(* POU RichThreePumpManager, CFC *)
FUNCTION_BLOCK RichThreePumpManager
VAR_INPUT
	start1: BOOL;
	start2: BOOL;
	p1main: BOOL;
	p2main: BOOL;
	p3main: BOOL;
	byCounter: BOOL;
	byWorkTime: BOOL;
	alarm1_in: BOOL;
	alarm2_in: BOOL;
	alarm3_in: BOOL;
	alarmReset: BOOL;
	start1man: BOOL;
	start2man: BOOL;
	start3man: BOOL;
	resetWTone: BOOL;
	resetWTtwo: BOOL;
	resetWTthree: BOOL;
	resetCounterOne: BOOL;
	resetCounterTwo: BOOL;
	resetCounterThree: BOOL;
	delayRepeatedStart: UINT;		(*задержка повторного пуска, сек.*)
	delayStart2: UINT;		(*задержка пуска второго после пуска первого, сек*)
END_VAR
VAR_OUTPUT
	p1mainActive: BOOL;
	p2mainActive: BOOL;
	p3mainActive: BOOL;
	byCounterActive: BOOL;
	byWTactive: BOOL;
	started1: BOOL;
	started2: BOOL;
	started3: BOOL;
	counterOne: UDINT;
	counterTwo: UDINT;
	counterThree: UDINT;
	days1: UINT;
	hours1: UINT;
	minutes1: UINT;
	seconds1: UINT;
	days2: UINT;
	hours2: UINT;
	minutes2: UINT;
	seconds2: UINT;
	days3: UINT;
	hours3: UINT;
	minutes3: UINT;
	seconds3: UINT;
	nextStartP1Timer: UINT;
	nextStartP2Timer: UINT;
	nextStartP3Timer: UINT;
	alarm1active: BOOL;
	alarm2active: BOOL;
	alarm3active: BOOL;
END_VAR
VAR
	ctpr: ChooseThreePumpRegime;
	slft: StartLessFromThree;
	alarmTrig1: RS;
	alarmTrig2: RS;
	alarmTrig3: RS;
	stp: SimpleThreePump;
	frsp1: FastRepeatedStartProtection;
	frsp2: FastRepeatedStartProtection;
	frsp3: FastRepeatedStartProtection;
	pps1: PulsePerSec;
	pps2: PulsePerSec;
	pps3: PulsePerSec;
	icwt1: ImpulsCounter;
	icw2: ImpulsCounter;
	icwt3: ImpulsCounter;
	ts1: TimeSeparator;
	ts2: TimeSeparator;
	ts3: TimeSeparator;
	ic1: ImpulsCounter;
	ic2: ImpulsCounter;
	ic3: ImpulsCounter;
	WorkTimeOne: UDINT;
	WorkTimeTwo: UDINT;
	WorkTimeThree: UDINT;
END_VAR
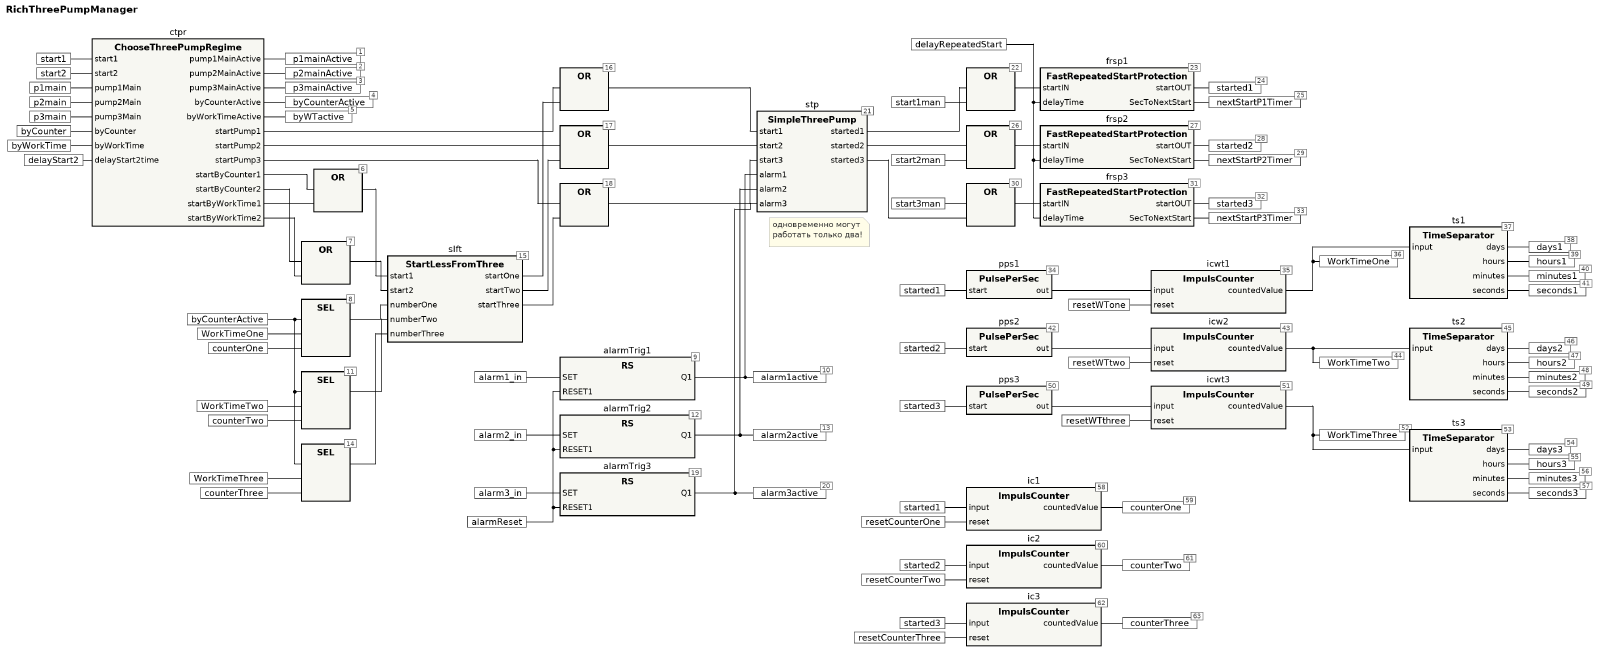
_CFC_ (* Continuous Function Chart, elements in execution order *)
(* одновременно могут / работать только два! *)
#0 ctpr:ChooseThreePumpRegime(start1: start1, start2: start2, pump1Main: p1main, pump2Main: p2main, pump3Main: p3main, byCounter: byCounter, byWorkTime: byWorkTime, delayStart2time: delayStart2)
#1 p1mainActive <= #0.pump1MainActive
#2 p2mainActive <= #0.pump2MainActive
#3 p3mainActive <= #0.pump3MainActive
#4 byCounterActive <= #0.byCounterActive
#5 byWTactive <= #0.byWorkTimeActive
#6 OR(#0.startByCounter1, #0.startByWorkTime1)
#7 OR(#0.startByCounter2, #0.startByWorkTime2)
#8 SEL(byCounterActive, WorkTimeOne, counterOne)
#9 alarmTrig1:RS(SET: alarm1_in, RESET1: alarmReset)
#10 alarm1active <= #9.Q1
#11 SEL(byCounterActive, WorkTimeTwo, counterTwo)
#12 alarmTrig2:RS(SET: alarm2_in, RESET1: alarmReset)
#13 alarm2active <= #12.Q1
#14 SEL(byCounterActive, WorkTimeThree, counterThree)
#15 slft:StartLessFromThree(start1: #6, start2: #7, numberOne: #8, numberTwo: #11, numberThree: #14)
#16 OR(#0.startPump1, #15.startOne)
#17 OR(#0.startPump2, #15.startTwo)
#18 OR(#0.startPump3, #15.startThree)
#19 alarmTrig3:RS(SET: alarm3_in, RESET1: alarmReset)
#20 alarm3active <= #19.Q1
#21 stp:SimpleThreePump(start1: #16, start2: #17, start3: #18, alarm1: #9.Q1, alarm2: #12.Q1, alarm3: #19.Q1)
#22 OR(#21.started1, start1man)
#23 frsp1:FastRepeatedStartProtection(startIN: #22, delayTime: delayRepeatedStart)
#24 started1 <= #23.startOUT
#25 nextStartP1Timer <= #23.SecToNextStart
#26 OR(#21.started2, start2man)
#27 frsp2:FastRepeatedStartProtection(startIN: #26, delayTime: delayRepeatedStart)
#28 started2 <= #27.startOUT
#29 nextStartP2Timer <= #27.SecToNextStart
#30 OR(start3man, #21.started3)
#31 frsp3:FastRepeatedStartProtection(startIN: #30, delayTime: delayRepeatedStart)
#32 started3 <= #31.startOUT
#33 nextStartP3Timer <= #31.SecToNextStart
#34 pps1:PulsePerSec(start: started1)
#35 icwt1:ImpulsCounter(input: #34.out, reset: resetWTone)
#36 WorkTimeOne <= #35.countedValue
#37 ts1:TimeSeparator(input: #35.countedValue)
#38 days1 <= #37.days
#39 hours1 <= #37.hours
#40 minutes1 <= #37.minutes
#41 seconds1 <= #37.seconds
#42 pps2:PulsePerSec(start: started2)
#43 icw2:ImpulsCounter(input: #42.out, reset: resetWTtwo)
#44 WorkTimeTwo <= #43.countedValue
#45 ts2:TimeSeparator(input: #43.countedValue)
#46 days2 <= #45.days
#47 hours2 <= #45.hours
#48 minutes2 <= #45.minutes
#49 seconds2 <= #45.seconds
#50 pps3:PulsePerSec(start: started3)
#51 icwt3:ImpulsCounter(input: #50.out, reset: resetWTthree)
#52 WorkTimeThree <= #51.countedValue
#53 ts3:TimeSeparator(input: #51.countedValue)
#54 days3 <= #53.days
#55 hours3 <= #53.hours
#56 minutes3 <= #53.minutes
#57 seconds3 <= #53.seconds
#58 ic1:ImpulsCounter(input: started1, reset: resetCounterOne)
#59 counterOne <= #58.countedValue
#60 ic2:ImpulsCounter(input: started2, reset: resetCounterTwo)
#61 counterTwo <= #60.countedValue
#62 ic3:ImpulsCounter(input: started3, reset: resetCounterThree)
#63 counterThree <= #62.countedValue
_END_CFC_
(* the same logic as Structured Text *)
(* одновременно могут / работать только два! *)
ctpr(start1 := start1, start2 := start2, pump1Main := p1main, pump2Main := p2main, pump3Main := p3main, byCounter := byCounter, byWorkTime := byWorkTime, delayStart2time := delayStart2);
p1mainActive := ctpr.pump1MainActive;
p2mainActive := ctpr.pump2MainActive;
p3mainActive := ctpr.pump3MainActive;
byCounterActive := ctpr.byCounterActive;
byWTactive := ctpr.byWorkTimeActive;
alarmTrig1(SET := alarm1_in, RESET1 := alarmReset);
alarm1active := alarmTrig1.Q1;
alarmTrig2(SET := alarm2_in, RESET1 := alarmReset);
alarm2active := alarmTrig2.Q1;
slft(start1 := ctpr.startByCounter1 OR ctpr.startByWorkTime1, start2 := ctpr.startByCounter2 OR ctpr.startByWorkTime2, numberOne := SEL(byCounterActive, WorkTimeOne, counterOne), numberTwo := SEL(byCounterActive, WorkTimeTwo, counterTwo), numberThree := SEL(byCounterActive, WorkTimeThree, counterThree));
alarmTrig3(SET := alarm3_in, RESET1 := alarmReset);
alarm3active := alarmTrig3.Q1;
stp(start1 := ctpr.startPump1 OR slft.startOne, start2 := ctpr.startPump2 OR slft.startTwo, start3 := ctpr.startPump3 OR slft.startThree, alarm1 := alarmTrig1.Q1, alarm2 := alarmTrig2.Q1, alarm3 := alarmTrig3.Q1);
frsp1(startIN := stp.started1 OR start1man, delayTime := delayRepeatedStart);
started1 := frsp1.startOUT;
nextStartP1Timer := frsp1.SecToNextStart;
frsp2(startIN := stp.started2 OR start2man, delayTime := delayRepeatedStart);
started2 := frsp2.startOUT;
nextStartP2Timer := frsp2.SecToNextStart;
frsp3(startIN := start3man OR stp.started3, delayTime := delayRepeatedStart);
started3 := frsp3.startOUT;
nextStartP3Timer := frsp3.SecToNextStart;
pps1(start := started1);
icwt1(input := pps1.out, reset := resetWTone);
WorkTimeOne := icwt1.countedValue;
ts1(input := icwt1.countedValue);
days1 := ts1.days;
hours1 := ts1.hours;
minutes1 := ts1.minutes;
seconds1 := ts1.seconds;
pps2(start := started2);
icw2(input := pps2.out, reset := resetWTtwo);
WorkTimeTwo := icw2.countedValue;
ts2(input := icw2.countedValue);
days2 := ts2.days;
hours2 := ts2.hours;
minutes2 := ts2.minutes;
seconds2 := ts2.seconds;
pps3(start := started3);
icwt3(input := pps3.out, reset := resetWTthree);
WorkTimeThree := icwt3.countedValue;
ts3(input := icwt3.countedValue);
days3 := ts3.days;
hours3 := ts3.hours;
minutes3 := ts3.minutes;
seconds3 := ts3.seconds;
ic1(input := started1, reset := resetCounterOne);
counterOne := ic1.countedValue;
ic2(input := started2, reset := resetCounterTwo);
counterTwo := ic2.countedValue;
ic3(input := started3, reset := resetCounterThree);
counterThree := ic3.countedValue;
END_FUNCTION_BLOCK

(* POU StartLessFromThree, ST *)
FUNCTION_BLOCK StartLessFromThree
VAR_INPUT
	start1: BOOL;
	start2: BOOL;
	numberOne: UDINT;
	numberTwo: UDINT;
	numberThree: UDINT;
END_VAR
VAR_OUTPUT
	startOne: BOOL;
	startTwo: BOOL;
	startThree: BOOL;
END_VAR
VAR
	flag1: BOOL := FALSE;
	flag2: BOOL := FALSE;
	starter: UINT;
END_VAR
IF start1 = TRUE THEN

	IF flag1= FALSE THEN

		IF numberOne  <=  numberTwo AND numberOne <= numberThree THEN
			starter := 0;
			flag1 := TRUE;
		END_IF
		
		IF flag1 = FALSE AND  numberTwo  <=  numberOne AND numberTwo <= numberThree THEN
			starter := 1;
			flag1 := TRUE;
		END_IF
		
		IF flag1 = FALSE AND numberThree  <=  numberOne AND numberThree <= numberTwo THEN
			starter := 2;
			flag1 := TRUE;
		END_IF

	END_IF

	CASE starter OF
		0: startOne := TRUE;
		1: startTwo := TRUE;
		2: startThree := TRUE;
	ELSE
		startOne := FALSE;
		startTwo := FALSE;
		startThree := FALSE;
	END_CASE

		IF start2 = TRUE THEN
			IF flag2 = FALSE THEN
				CASE starter OF
					0:   IF numberTwo <= numberThree THEN
							startTwo := TRUE;
							flag2 := TRUE;
						ELSE
							startThree := TRUE;
							flag2 := TRUE;
						END_IF
					1:   IF numberOne <= numberThree THEN
							startOne := TRUE;
							flag2 := TRUE;
						ELSE
							startThree := TRUE;
							flag2 := TRUE;
						END_IF
					2:   IF numberOne <= numberTwo THEN
							startOne := TRUE;
							flag2 := TRUE;
						ELSE
							startTwo := TRUE;
							flag2 := TRUE;
						END_IF
				END_CASE
			END_IF
		ELSE
			CASE starter OF
				0:   startOne := TRUE;
					startTwo := FALSE;
					startThree := FALSE;
					flag2 := FALSE;
				1:   startTwo := TRUE;
					startOne := FALSE;
					startThree := FALSE;
					flag2 := FALSE;
				2:   startThree := TRUE;
					startOne := FALSE;
					startTwo := FALSE;
					flag2 := FALSE;
			ELSE
				startOne := FALSE;
				startTwo := FALSE;
				startThree := FALSE;
	END_CASE
		END_IF

ELSE

		startOne := FALSE;
		startTwo := FALSE;
		startThree := FALSE;
		flag1 := FALSE;

END_IF
END_FUNCTION_BLOCK

(* POU SimpleThreePump, CFC *)
FUNCTION_BLOCK SimpleThreePump
VAR_INPUT
	start1: BOOL; (*сигнал на пуск насоса 1*)
	start2: BOOL; (*сигнал на пуск насоса 2*)
	start3: BOOL; (*сигнал на пуск насоса 3*)
	alarm1: BOOL; (*авария насоса 1*)
	alarm2: BOOL; (*авария насоса 2*)
	alarm3: BOOL; (*авария насоса 3*)
END_VAR
VAR_OUTPUT
	started1: BOOL; (*сигнал на запуск насоса 1*)
	started2: BOOL; (*сигнал на запуск насоса 2*)
	started3: BOOL; (*сигнал на запуск насоса 3*)
END_VAR
VAR
	pump1changer: BOOL;
	pump2changer: BOOL;
	pump3changer: BOOL;
END_VAR
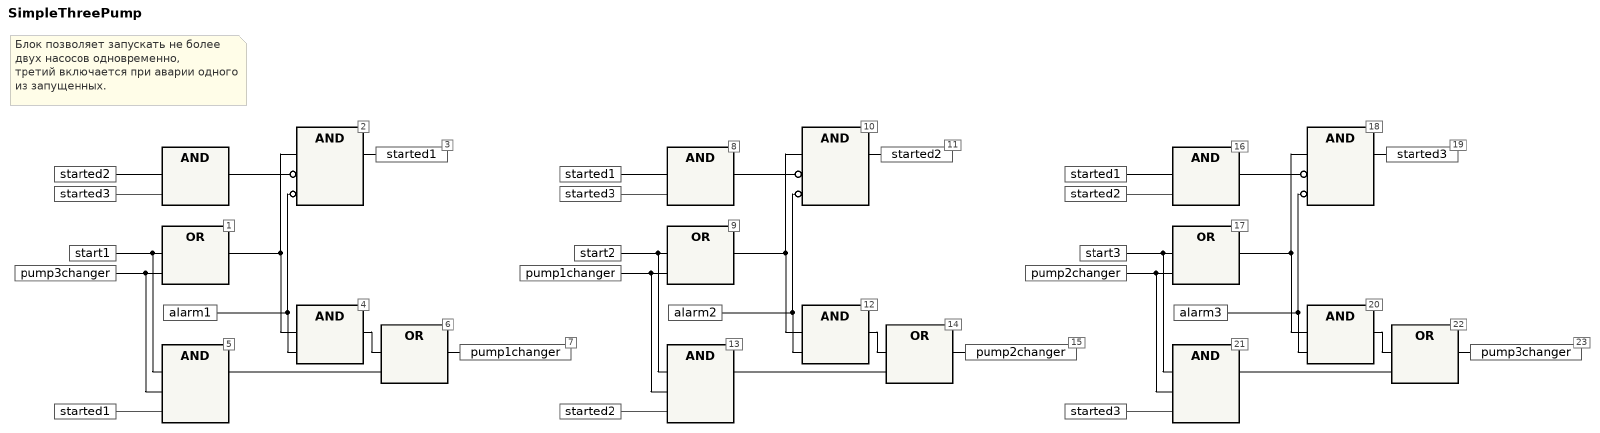
_CFC_ (* Continuous Function Chart, elements in execution order *)
#0 AND(started2, started3)
#1 OR(start1, pump3changer)
(* Блок позволяет запускать не более / двух насосов одновременно, / третий включается при аварии одного / из запущенных. *)
#2 AND(#1, NOT #0, NOT alarm1)
#3 started1 <= #2
#4 AND(#1, alarm1)
#5 AND(start1, pump3changer, started1)
#6 OR(#4, #5)
#7 pump1changer <= #6
#8 AND(started1, started3)
#9 OR(start2, pump1changer)
#10 AND(#9, NOT #8, NOT alarm2)
#11 started2 <= #10
#12 AND(#9, alarm2)
#13 AND(start2, pump1changer, started2)
#14 OR(#12, #13)
#15 pump2changer <= #14
#16 AND(started1, started2)
#17 OR(start3, pump2changer)
#18 AND(#17, NOT #16, NOT alarm3)
#19 started3 <= #18
#20 AND(#17, alarm3)
#21 AND(start3, pump2changer, started3)
#22 OR(#20, #21)
#23 pump3changer <= #22
_END_CFC_
(* the same logic as Structured Text *)
(* Блок позволяет запускать не более / двух насосов одновременно, / третий включается при аварии одного / из запущенных. *)
started1 := (start1 OR pump3changer) AND NOT (started2 AND started3) AND NOT alarm1;
pump1changer := ((start1 OR pump3changer) AND alarm1) OR (start1 AND pump3changer AND started1);
started2 := (start2 OR pump1changer) AND NOT (started1 AND started3) AND NOT alarm2;
pump2changer := ((start2 OR pump1changer) AND alarm2) OR (start2 AND pump1changer AND started2);
started3 := (start3 OR pump2changer) AND NOT (started1 AND started2) AND NOT alarm3;
pump3changer := ((start3 OR pump2changer) AND alarm3) OR (start3 AND pump2changer AND started3);
END_FUNCTION_BLOCK

(* POU TimeSeparator, ST *)
FUNCTION_BLOCK TimeSeparator
VAR_INPUT
	 input: UDINT; (*Вход счетчика  наработки и т.п., сек.*)
END_VAR
VAR_OUTPUT
	days: UINT; (*Выход наработка, дней*)
	hours: UINT; (*Выход наработка, часов*)
	minutes: UINT; (*Выход наработка, минут*)
	seconds: UINT; (*Выход наработка, секунд*)
END_VAR
VAR
	temp: UDINT;
END_VAR
days:= UDINT_TO_INT (input / (60 * 60 * 24));
temp:= input MOD (60 * 60 * 24);
hours:= UDINT_TO_INT (temp / (60 * 60));
temp:= temp MOD (60 * 60);
minutes:= UDINT_TO_INT (temp / 60);
temp:= temp MOD 60;
seconds:= UDINT_TO_INT (temp);
END_FUNCTION_BLOCK

(* POU RichTwoPumpManager, CFC *)
FUNCTION_BLOCK RichTwoPumpManager
VAR_INPUT
	start: BOOL;		(*Сигнал на запуск насоса согласно выбранному режиму.*)
	setPump1main: BOOL;		(*Установить режим - насос 1 = главный.
Включать импульсом.*)
	setPump2main: BOOL;		(*Установить режим - насос 2 = главный.
Включать импульсом.*)
	setByCounter: BOOL;		(*Установить режим - по количеству включений.
Включать импульсом.*)
	setByWorkTime: BOOL;		(*Установить режим - по наработке.
Включать импульсом.*)
	resetPump1counter: BOOL;		(*Сброс счетчика количества включений насоса 1.*)
	resetPump2counter: BOOL;		(*Сброс счетчика количества включений насоса 2.*)
	resetWorkTimePump1: BOOL;		(*Сброс счетчика наработки насоса 1.*)
	resetWorkTimePump2: BOOL;		(*Сброс счетчика наработки насоса 2.*)
	startPump1man: BOOL;		(*Пуск насоса 1 вручную независимо от текущего режима.*)
	startPump2man: BOOL;		(*Пуск насоса 2 вручную независимо от текущего режима.*)
	stop: BOOL;		(*Стоп обоих насосов пока вход активен.
Не стоит применять для штатного останова.*)
	resetAlarms: BOOL;		(*Сброс аварий насоса.*)
	delayRepeatedStartTime: WORD;		(*Количество секунд на задержку повторного пуска насоса.
Защита от частых включений. Если ничего не подключено = 300сек.*)
	alarmPump1input: BOOL;		(*Вход от источника сигнала об аварии насоса 1.*)
	alarmPump2input: BOOL;		(*Вход от источника сигнала об аварии насоса 2.*)
END_VAR
VAR_OUTPUT
	regimePump1Main: BOOL;		(*Текущий режим - насос 1 = главный.*)
	regimePump2Main: BOOL;		(*Текущий режим - насос 2 = главный.*)
	regimeByCounter: BOOL;		(*Текущий режим - по количеству включений.*)
	regimeByWorkTime: BOOL;		(*Текущий режим - по наработке.*)
	counterPump1: DWORD;		(*Количество включений насоса 1.*)
	counterPump2: DWORD;		(*Количество включений насоса 2.*)
	daysPump1: WORD;		(*Количество отработанных дней насоса 1.*)
	hoursPump1: WORD;		(*Количество отработанных часов насоса 1.*)
	minutesPump1: WORD;		(*Количество отработанных минут насоса 1.*)
	secondsPump1: WORD;		(*Количество отработанных секунд насоса 1.*)
	daysPump2: WORD;		(*Количество отработанных дней насоса 2.*)
	hoursPump2: WORD;		(*Количество отработанных часов насоса 2.*)
	minutesPump2: WORD;		(*Количество отработанных минут насоса 2.*)
	secondsPump2: WORD;		(*Количество отработанных секунд насоса 2.*)
	pump1starter: BOOL;		(*Сигнал на запуск насоса 1.*)
	pump2starter: BOOL;		(*Сигнал на запуск насоса 2.*)
	nextStartP1timer: WORD;		(*Обратный отсчет до возможности повторного пуска насоса 1.*)
	nextStartP2timer: WORD;		(*Обратный отсчет до возможности повторного пуска насоса 2.*)
	alarmPump1output: BOOL;		(*Сигнал авария насоса 1.
Триггерится, нужен сброс.*)
	alarmPump2output: BOOL;		(*Сигнал авария насоса 2.
Триггерится, нужен сброс.*)
END_VAR
VAR
	ChoosePumpRegime: ChoosePumpRegime;		(*Блок выбора режима включения.*)
	CounterManager: CounterManager;		(*Блок выбора и запуска насоса по наработке.*)
	WorkTimeManager: WorkTimeManager;		(*Блок выбора и запуска насоса с меньшей наработкой.*)
	simpleTimeManager: SimpleTwoPumpManager;		(*Блок управления двумя насосами, горячий резерв, автоматическое переключение.*)
END_VAR
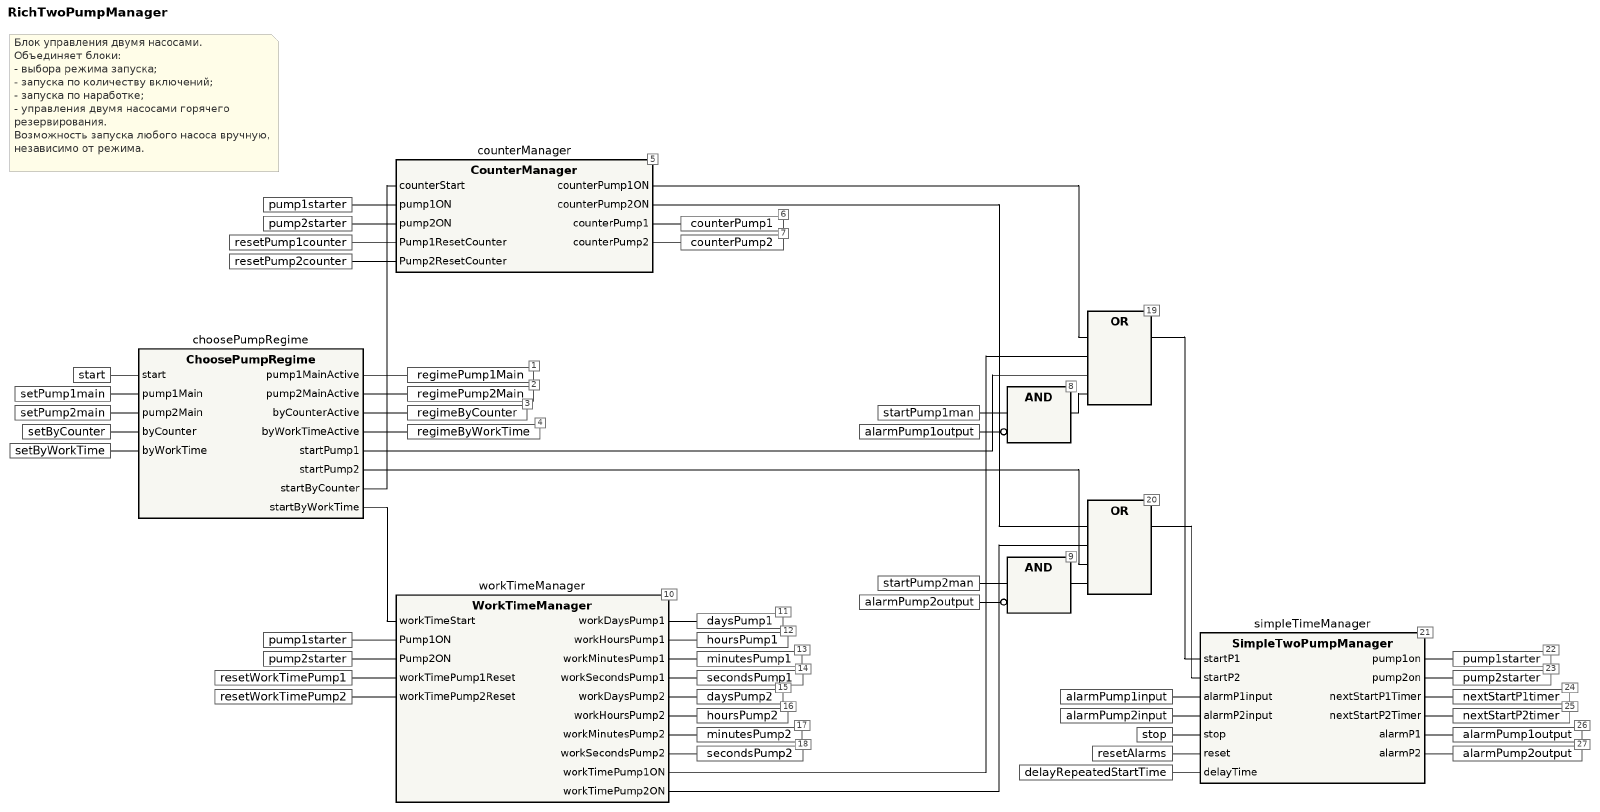
_CFC_ (* Continuous Function Chart, elements in execution order *)
(* Блок управления двумя насосами. / Объединяет блоки: / - выбора режима запуска; / - запуска по количеству включений; / - запуска по наработке; / - управления двумя насосами горячего резервирования. / Возможность запуска любого насоса вручную, / независимо от режима. *)
#0 choosePumpRegime:ChoosePumpRegime(start: start, pump1Main: setPump1main, pump2Main: setPump2main, byCounter: setByCounter, byWorkTime: setByWorkTime)
#1 regimePump1Main <= #0.pump1MainActive
#2 regimePump2Main <= #0.pump2MainActive
#3 regimeByCounter <= #0.byCounterActive
#4 regimeByWorkTime <= #0.byWorkTimeActive
#5 counterManager:CounterManager(counterStart: #0.startByCounter, pump1ON: pump1starter, pump2ON: pump2starter, Pump1ResetCounter: resetPump1counter, Pump2ResetCounter: resetPump2counter)
#6 counterPump1 <= #5.counterPump1
#7 counterPump2 <= #5.counterPump2
#8 AND(startPump1man, NOT alarmPump1output)
#9 AND(startPump2man, NOT alarmPump2output)
#10 workTimeManager:WorkTimeManager(workTimeStart: #0.startByWorkTime, Pump1ON: pump1starter, Pump2ON: pump2starter, workTimePump1Reset: resetWorkTimePump1, workTimePump2Reset: resetWorkTimePump2)
#11 daysPump1 <= #10.workDaysPump1
#12 hoursPump1 <= #10.workHoursPump1
#13 minutesPump1 <= #10.workMinutesPump1
#14 secondsPump1 <= #10.workSecondsPump1
#15 daysPump2 <= #10.workDaysPump2
#16 hoursPump2 <= #10.workHoursPump2
#17 minutesPump2 <= #10.workMinutesPump2
#18 secondsPump2 <= #10.workSecondsPump2
#19 OR(#5.counterPump1ON, #10.workTimePump1ON, #0.startPump1, #8)
#20 OR(#5.counterPump2ON, #10.workTimePump2ON, #0.startPump2, #9)
#21 simpleTimeManager:SimpleTwoPumpManager(startP1: #19, startP2: #20, alarmP1input: alarmPump1input, alarmP2input: alarmPump2input, stop: stop, reset: resetAlarms, delayTime: delayRepeatedStartTime)
#22 pump1starter <= #21.pump1on
#23 pump2starter <= #21.pump2on
#24 nextStartP1timer <= #21.nextStartP1Timer
#25 nextStartP2timer <= #21.nextStartP2Timer
#26 alarmPump1output <= #21.alarmP1
#27 alarmPump2output <= #21.alarmP2
_END_CFC_
(* the same logic as Structured Text *)
(* Блок управления двумя насосами. / Объединяет блоки: / - выбора режима запуска; / - запуска по количеству включений; / - запуска по наработке; / - управления двумя насосами горячего резервирования. / Возможность запуска любого насоса вручную, / независимо от режима. *)
choosePumpRegime(start := start, pump1Main := setPump1main, pump2Main := setPump2main, byCounter := setByCounter, byWorkTime := setByWorkTime);
regimePump1Main := choosePumpRegime.pump1MainActive;
regimePump2Main := choosePumpRegime.pump2MainActive;
regimeByCounter := choosePumpRegime.byCounterActive;
regimeByWorkTime := choosePumpRegime.byWorkTimeActive;
counterManager(counterStart := choosePumpRegime.startByCounter, pump1ON := pump1starter, pump2ON := pump2starter, Pump1ResetCounter := resetPump1counter, Pump2ResetCounter := resetPump2counter);
counterPump1 := counterManager.counterPump1;
counterPump2 := counterManager.counterPump2;
workTimeManager(workTimeStart := choosePumpRegime.startByWorkTime, Pump1ON := pump1starter, Pump2ON := pump2starter, workTimePump1Reset := resetWorkTimePump1, workTimePump2Reset := resetWorkTimePump2);
daysPump1 := workTimeManager.workDaysPump1;
hoursPump1 := workTimeManager.workHoursPump1;
minutesPump1 := workTimeManager.workMinutesPump1;
secondsPump1 := workTimeManager.workSecondsPump1;
daysPump2 := workTimeManager.workDaysPump2;
hoursPump2 := workTimeManager.workHoursPump2;
minutesPump2 := workTimeManager.workMinutesPump2;
secondsPump2 := workTimeManager.workSecondsPump2;
simpleTimeManager(startP1 := counterManager.counterPump1ON OR workTimeManager.workTimePump1ON OR choosePumpRegime.startPump1 OR (startPump1man AND NOT alarmPump1output), startP2 := counterManager.counterPump2ON OR workTimeManager.workTimePump2ON OR choosePumpRegime.startPump2 OR (startPump2man AND NOT alarmPump2output), alarmP1input := alarmPump1input, alarmP2input := alarmPump2input, stop := stop, reset := resetAlarms, delayTime := delayRepeatedStartTime);
pump1starter := simpleTimeManager.pump1on;
pump2starter := simpleTimeManager.pump2on;
nextStartP1timer := simpleTimeManager.nextStartP1Timer;
nextStartP2timer := simpleTimeManager.nextStartP2Timer;
alarmPump1output := simpleTimeManager.alarmP1;
alarmPump2output := simpleTimeManager.alarmP2;
END_FUNCTION_BLOCK

(* POU WorkTimeManager, CFC *)
FUNCTION_BLOCK WorkTimeManager
VAR
	workTimePump1: TimeSeparator;		(*Блок вывода времени наработки  насоса 1.*)
	workTimePump2: TimeSeparator;		(*Блок вывода времени наработки насоса 2.*)
	currentWorkTimePump1: DWORD;		(*Текущая наработка в секундах насоса 1.*)
	currentWorkTimePump2: DWORD;		(*Текущая наработка в секундах насоса 2.*)
	pulsarP1: PulsePerSec;		(*Генератор импульса в секунду для наработки насоса 1.*)
	pulsarP2: PulsePerSec;		(*Генератор импульса в секунду для наработки насоса 2.*)
	timeStartRtrig: R_TRIG;		(*Детектор переднего фронта сигнала на запуск.*)
	timeStartFtrig: F_TRIG;		(*Детектор спада сигнала на запуск.*)
	RStrigTimePump1: RS;		(*RSтриггер сигнала на запуск насоса 1.*)
	RStrigTimePump2: RS;		(*RSтриггер сигнала на запуск насоса 2.*)
END_VAR
VAR_OUTPUT
	workDaysPump1: WORD;		(*Количество отработанных дней для насоса 1.*)
	workHoursPump1: WORD;		(*Количество отработанных часов для насоса 1.*)
	workMinutesPump1: WORD;		(*Количество отработанных минут для насоса 1.*)
	workSecondsPump1: WORD;		(*Количество отработанных секунд для насоса 1.*)
	workDaysPump2: WORD;		(*Количество отработанных дней для насоса 2.*)
	workHoursPump2: WORD;		(*Количество отработанных часов для насоса 2.*)
	workMinutesPump2: WORD;		(*Количество отработанных минут для насоса 2.*)
	workSecondsPump2: WORD;		(*Количество отработанных секунд для насоса 2.*)
	workTimePump1ON: BOOL;		(*Выход на запуск насоса 1.*)
	workTimePump2ON: BOOL;		(*Выход на запуск насоса 2.*)
END_VAR
VAR_INPUT
	workTimeStart: BOOL;		(*Сигнал на запуск насоса с наименьшим временем работы.*)
	Pump1ON: BOOL;		(*Сигнал подтверждение о запуске насоса 1.*)
	Pump2ON: BOOL;		(*Сигнал подтверждение о запуске насоса 2.*)
	workTimePump1Reset: BOOL;		(*Сброс времени наработки насоса 1.*)
	workTimePump2Reset: BOOL;		(*Сброс времени наработки насоса 2.*)
END_VAR
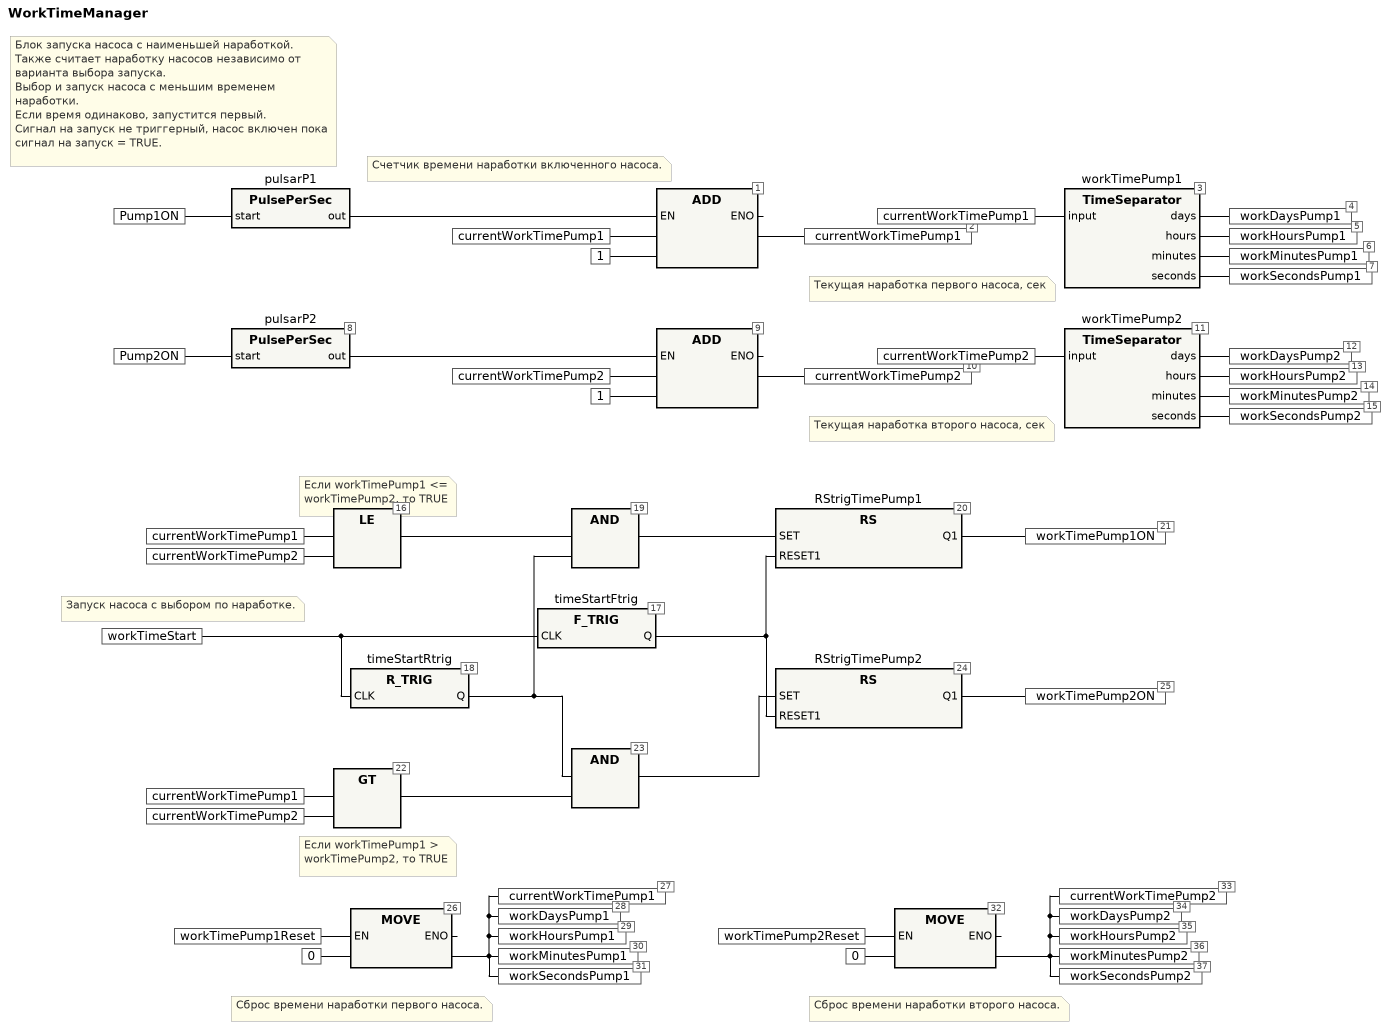
_CFC_ (* Continuous Function Chart, elements in execution order *)
(* Текущая наработка второго насоса, сек *)
(* Сброс времени наработки второго насоса. *)
(* Текущая наработка первого насоса, сек *)
(* Счетчик времени наработки включенного насоса. *)
(* Если workTimePump1 > / workTimePump2, то TRUE *)
(* Если workTimePump1 <= / workTimePump2, то TRUE *)
(* Запуск насоса с выбором по наработке. *)
(* Блок запуска насоса с наименьшей наработкой. / Также считает наработку насосов независимо от варианта выбора запуска. / Выбор и запуск насоса с меньшим временем наработки. / Если время одинаково, запустится первый. / Сигнал на запуск не триггерный, насос включен пока сигнал на запуск = TRUE. *)
(* Сброс времени наработки первого насоса. *)
#0 pulsarP1:PulsePerSec(start: Pump1ON)
#1 ADD(EN: #0.out, currentWorkTimePump1, 1)
#2 currentWorkTimePump1 <= #1
#3 workTimePump1:TimeSeparator(input: currentWorkTimePump1)
#4 workDaysPump1 <= #3.days
#5 workHoursPump1 <= #3.hours
#6 workMinutesPump1 <= #3.minutes
#7 workSecondsPump1 <= #3.seconds
#8 pulsarP2:PulsePerSec(start: Pump2ON)
#9 ADD(EN: #8.out, currentWorkTimePump2, 1)
#10 currentWorkTimePump2 <= #9
#11 workTimePump2:TimeSeparator(input: currentWorkTimePump2)
#12 workDaysPump2 <= #11.days
#13 workHoursPump2 <= #11.hours
#14 workMinutesPump2 <= #11.minutes
#15 workSecondsPump2 <= #11.seconds
#16 LE(currentWorkTimePump1, currentWorkTimePump2)
#17 timeStartFtrig:F_TRIG(CLK: workTimeStart)
#18 timeStartRtrig:R_TRIG(CLK: workTimeStart)
#19 AND(#16, #18.Q)
#20 RStrigTimePump1:RS(SET: #19, RESET1: #17.Q)
#21 workTimePump1ON <= #20.Q1
#22 GT(currentWorkTimePump1, currentWorkTimePump2)
#23 AND(#18.Q, #22)
#24 RStrigTimePump2:RS(SET: #23, RESET1: #17.Q)
#25 workTimePump2ON <= #24.Q1
#26 MOVE(EN: workTimePump1Reset, 0)
#27 currentWorkTimePump1 <= #26
#28 workDaysPump1 <= #26
#29 workHoursPump1 <= #26
#30 workMinutesPump1 <= #26
#31 workSecondsPump1 <= #26
#32 MOVE(EN: workTimePump2Reset, 0)
#33 currentWorkTimePump2 <= #32
#34 workDaysPump2 <= #32
#35 workHoursPump2 <= #32
#36 workMinutesPump2 <= #32
#37 workSecondsPump2 <= #32
_END_CFC_
END_FUNCTION_BLOCK

(* POU SimpleTwoPumpManager, CFC *)
FUNCTION_BLOCK SimpleTwoPumpManager

VAR
	alarmP1trig: RS;		(*Триггер - защелка аварии насоса 1.*)
	alarmP2trig: RS;		(*Триггер - защелка аварии насоса 2.*)
	stopPump1Detector: F_TRIG;		(*Детектор спада сигнала (останов) насоса 1.*)
	stopPump2Detector: F_TRIG;		(*Детектор спада сигнала (останов) насоса 2.*)
	delayAfterStopP2: TOF;		(*Таймер задержки на включение
насоса 1 после останова насоса 2.*)
	delayAfterStopP1: TOF;		(*Таймер задержки на включение
насоса 2 после останова насоса 1.*)
	antiFreqStartPump1: TOF;		(*Таймер - предохранитель от частых пусков насоса 1.*)
	antiFreqStartPump2: TOF;		(*Таймер - предохранитель от частых пусков насоса 2.*)
	startPump1Trig: RS;		(*RS триггер на пуск насоса 1.*)
	startPump2Trig: RS;		(*RS триггер на пуск насоса 2.*)
	stopPump1: F_TRIG;		(*Сигнал на останов насоса 1.*)
	stopPump2: F_TRIG;		(*Сигнал на останов насоса 2.*)
END_VAR
VAR_INPUT
	startP1: BOOL;		(*Сигнал на запуск насоса 1.
Активен - пуск, неактивен - стоп.*)
	startP2: BOOL;		(*Сигнал на запуск насоса 2.
Активен - пуск, неактивен - стоп.*)
	alarmP1input: BOOL;		(*Сигнал авария от насоса 1.*)
	alarmP2input: BOOL;		(*Сигнал авария от насоса 2.*)
	stop: BOOL;		(*Сигнал на останов. Пока активен - пусков нет.
Общий на оба насоса.*)
	reset: BOOL;		(*Сброс аварий.*)
	delayTime: WORD := 300;		(*Задержка на повторный пуск в секундах.
Если ко входу ничего не подключено, то 300сек.*)
END_VAR
VAR_OUTPUT
	pump1on: BOOL;		(*Выход на запуск насоса 1.*)
	pump2on: BOOL;		(*Выход на запуск насоса 2.*)
	nextStartP1Timer: WORD;		(*Счетчик секунд до возможности повторного пуска насоса 1.*)
	nextStartP2Timer: WORD;		(*Счетчик секунд до возможности повторного пуска насоса 2.*)
	alarmP1: BOOL;		(*Статус - авария насоса 1.*)
	alarmP2: BOOL;		(*Статус - авария насоса 2.*)
END_VAR
VAR (* helpers for the ST form of the networks *)
	_t203 : TIME;
END_VAR
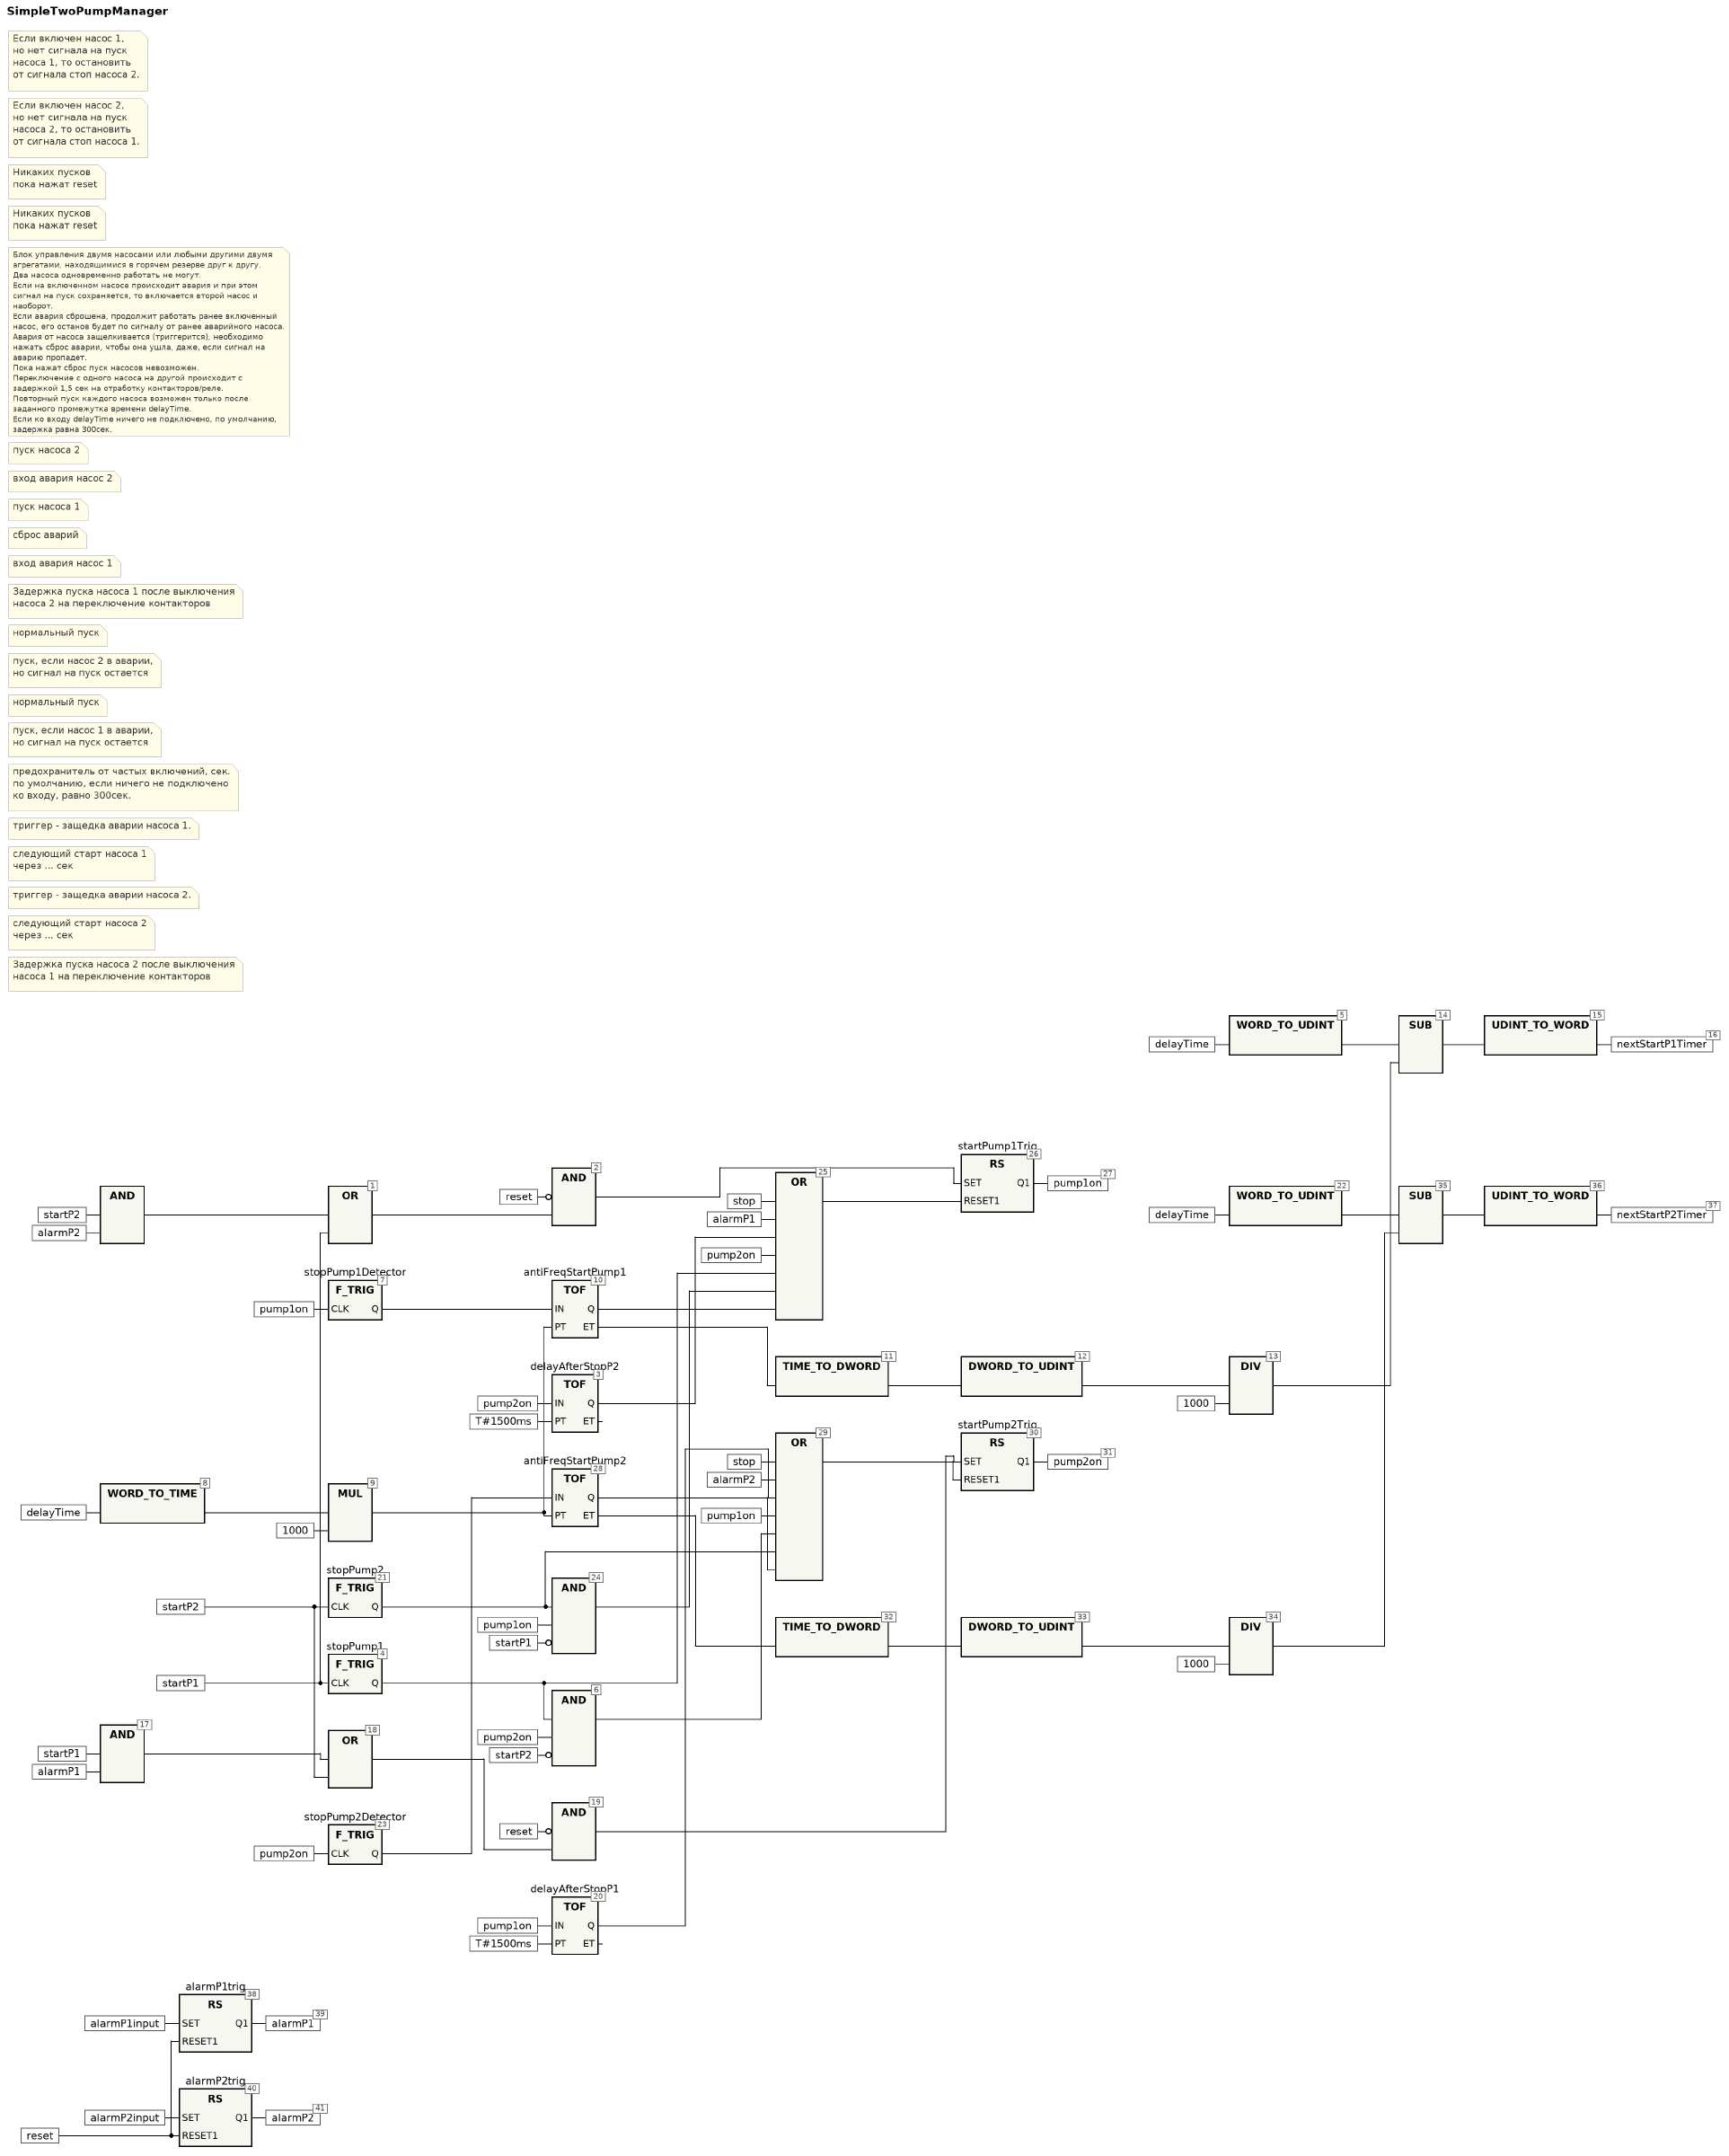
_CFC_ (* Continuous Function Chart, elements in execution order *)
(* Если включен насос 1, / но нет сигнала на пуск / насоса 1, то остановить / от сигнала стоп насоса 2. *)
(* Если включен насос 2, / но нет сигнала на пуск / насоса 2, то остановить / от сигнала стоп насоса 1. *)
(* Никаких пусков / пока нажат reset *)
(* Никаких пусков / пока нажат reset *)
(* Блок управления двумя насосами или любыми другими двумя агрегатами, находящимися в горячем резерве друг к другу. / Два насоса одновременно работать не могут. / Если на включенном насосе происходит авария и при этом сигнал на пуск сохраняется, то включается второй насос и наоборот. / Если авария сброшена, продолжит работать ранее включенный насос, его останов будет по сигналу от ранее аварийного насоса. / Авария от насоса защелкивается (триггерится), необходимо нажать сброс аварии, чтобы она ушла, даже, если сигнал на аварию пропадет. / Пока нажат сброс пуск насосов невозможен. / Переключение с одного насоса на другой происходит с задержкой 1,5 сек на отработку контакторов/реле. / Повторный пуск каждого насоса возможен только после заданного промежутка времени delayTime. / Если ко входу delayTime ничего не подключено, по умолчанию, задержка равна 300сек. *)
(* пуск насоса 2 *)
(* вход авария насос 2 *)
(* пуск насоса 1 *)
(* сброс аварий *)
(* вход авария насос 1 *)
(* Задержка пуска насоса 1 после выключения / насоса 2 на переключение контакторов *)
(* нормальный пуск *)
(* пуск, если насос 2 в аварии, / но сигнал на пуск остается *)
(* нормальный пуск *)
(* пуск, если насос 1 в аварии, / но сигнал на пуск остается *)
(* предохранитель от частых включений, сек. / по умолчанию, если ничего не подключено / ко входу, равно 300сек. *)
(* триггер - защедка аварии насоса 1. *)
(* cледующий старт насоса 1 / через ... сек *)
(* триггер - защедка аварии насоса 2. *)
(* cледующий старт насоса 2 / через ... сек *)
(* Задержка пуска насоса 2 после выключения / насоса 1 на переключение контакторов *)
#0 AND(startP2, alarmP2)
#1 OR(#0, startP1)
#2 AND(NOT reset, #1)
#3 delayAfterStopP2:TOF(IN: pump2on, PT: T#1500ms)
#4 stopPump1:F_TRIG(CLK: startP1)
#5 WORD_TO_UDINT(delayTime)
#6 AND(#4.Q, pump2on, NOT startP2)
#7 stopPump1Detector:F_TRIG(CLK: pump1on)
#8 WORD_TO_TIME(delayTime)
#9 MUL(#8, 1000)
#10 antiFreqStartPump1:TOF(IN: #7.Q, PT: #9)
#11 TIME_TO_DWORD(#10.ET)
#12 DWORD_TO_UDINT(#11)
#13 DIV(#12, 1000)
#14 SUB(#5, #13)
#15 UDINT_TO_WORD(#14)
#16 nextStartP1Timer <= #15
#17 AND(startP1, alarmP1)
#18 OR(#17, startP2)
#19 AND(NOT reset, #18)
#20 delayAfterStopP1:TOF(IN: pump1on, PT: T#1500ms)
#21 stopPump2:F_TRIG(CLK: startP2)
#22 WORD_TO_UDINT(delayTime)
#23 stopPump2Detector:F_TRIG(CLK: pump2on)
#24 AND(#21.Q, pump1on, NOT startP1)
#25 OR(stop, alarmP1, #3.Q, pump2on, #4.Q, #24, #10.Q)
#26 startPump1Trig:RS(SET: #2, RESET1: #25)
#27 pump1on <= #26.Q1
#28 antiFreqStartPump2:TOF(IN: #23.Q, PT: #9)
#29 OR(stop, alarmP2, #20.Q, pump1on, #6, #21.Q, #28.Q)
#30 startPump2Trig:RS(SET: #19, RESET1: #29)
#31 pump2on <= #30.Q1
#32 TIME_TO_DWORD(#28.ET)
#33 DWORD_TO_UDINT(#32)
#34 DIV(#33, 1000)
#35 SUB(#22, #34)
#36 UDINT_TO_WORD(#35)
#37 nextStartP2Timer <= #36
#38 alarmP1trig:RS(SET: alarmP1input, RESET1: reset)
#39 alarmP1 <= #38.Q1
#40 alarmP2trig:RS(SET: alarmP2input, RESET1: reset)
#41 alarmP2 <= #40.Q1
_END_CFC_
(* the same logic as Structured Text *)
(* Если включен насос 1, / но нет сигнала на пуск / насоса 1, то остановить / от сигнала стоп насоса 2. *)
(* Если включен насос 2, / но нет сигнала на пуск / насоса 2, то остановить / от сигнала стоп насоса 1. *)
(* Никаких пусков / пока нажат reset *)
(* Никаких пусков / пока нажат reset *)
(* Блок управления двумя насосами или любыми другими двумя агрегатами, находящимися в горячем резерве друг к другу. / Два насоса одновременно работать не могут. / Если на включенном насосе происходит авария и при этом сигнал на пуск сохраняется, то включается второй насос и наоборот. / Если авария сброшена, продолжит работать ранее включенный насос, его останов будет по сигналу от ранее аварийного насоса. / Авария от насоса защелкивается (триггерится), необходимо нажать сброс аварии, чтобы она ушла, даже, если сигнал на аварию пропадет. / Пока нажат сброс пуск насосов невозможен. / Переключение с одного насоса на другой происходит с задержкой 1,5 сек на отработку контакторов/реле. / Повторный пуск каждого насоса возможен только после заданного промежутка времени delayTime. / Если ко входу delayTime ничего не подключено, по умолчанию, задержка равна 300сек. *)
(* пуск насоса 2 *)
(* вход авария насос 2 *)
(* пуск насоса 1 *)
(* сброс аварий *)
(* вход авария насос 1 *)
(* Задержка пуска насоса 1 после выключения / насоса 2 на переключение контакторов *)
(* нормальный пуск *)
(* пуск, если насос 2 в аварии, / но сигнал на пуск остается *)
(* нормальный пуск *)
(* пуск, если насос 1 в аварии, / но сигнал на пуск остается *)
(* предохранитель от частых включений, сек. / по умолчанию, если ничего не подключено / ко входу, равно 300сек. *)
(* триггер - защедка аварии насоса 1. *)
(* cледующий старт насоса 1 / через ... сек *)
(* триггер - защедка аварии насоса 2. *)
(* cледующий старт насоса 2 / через ... сек *)
(* Задержка пуска насоса 2 после выключения / насоса 1 на переключение контакторов *)
delayAfterStopP2(IN := pump2on, PT := T#1500ms);
stopPump1(CLK := startP1);
stopPump1Detector(CLK := pump1on);
_t203 := WORD_TO_TIME(delayTime) * 1000;
antiFreqStartPump1(IN := stopPump1Detector.Q, PT := _t203);
nextStartP1Timer := UDINT_TO_WORD(WORD_TO_UDINT(delayTime) - (DWORD_TO_UDINT(TIME_TO_DWORD(antiFreqStartPump1.ET)) / 1000));
delayAfterStopP1(IN := pump1on, PT := T#1500ms);
stopPump2(CLK := startP2);
stopPump2Detector(CLK := pump2on);
startPump1Trig(SET := NOT reset AND ((startP2 AND alarmP2) OR startP1), RESET1 := stop OR alarmP1 OR delayAfterStopP2.Q OR pump2on OR stopPump1.Q OR (stopPump2.Q AND pump1on AND NOT startP1) OR antiFreqStartPump1.Q);
pump1on := startPump1Trig.Q1;
antiFreqStartPump2(IN := stopPump2Detector.Q, PT := _t203);
startPump2Trig(SET := NOT reset AND ((startP1 AND alarmP1) OR startP2), RESET1 := stop OR alarmP2 OR delayAfterStopP1.Q OR pump1on OR (stopPump1.Q AND pump2on AND NOT startP2) OR stopPump2.Q OR antiFreqStartPump2.Q);
pump2on := startPump2Trig.Q1;
nextStartP2Timer := UDINT_TO_WORD(WORD_TO_UDINT(delayTime) - (DWORD_TO_UDINT(TIME_TO_DWORD(antiFreqStartPump2.ET)) / 1000));
alarmP1trig(SET := alarmP1input, RESET1 := reset);
alarmP1 := alarmP1trig.Q1;
alarmP2trig(SET := alarmP2input, RESET1 := reset);
alarmP2 := alarmP2trig.Q1;
END_FUNCTION_BLOCK

(* POU TwoPumpOneDriveManager, CFC *)
FUNCTION_BLOCK TwoPumpOneDriveManager
	VAR_INPUT
	start: BOOL;		(*Сигнал на запуск насоса согласно выбранному режиму.*)
	setPump1main: BOOL;		(*Установить режим - насос 1 = главный.
Включать импульсом.*)
	setPump2main: BOOL;		(*Установить режим - насос 2 = главный.
Включать импульсом.*)
	setByCounter: BOOL;		(*Установить режим - по количеству включений.
Включать импульсом.*)
	setByWorkTime: BOOL;		(*Установить режим - по наработке.
Включать импульсом.*)
	resetPump1counter: BOOL;		(*Сброс счетчика количества включений насоса 1.*)
	resetPump2counter: BOOL;		(*Сброс счетчика количества включений насоса 2.*)
	resetWorkTimePump1: BOOL;		(*Сброс счетчика наработки насоса 1.*)
	resetWorkTimePump2: BOOL;		(*Сброс счетчика наработки насоса 2.*)
	startPump1man: BOOL;		(*Пуск насоса 1 вручную независимо от текущего режима.*)
	startPump2man: BOOL;		(*Пуск насоса 2 вручную независимо от текущего режима.*)
	stop: BOOL;		(*Стоп обоих насосов пока вход активен.
Не стоит применять для штатного останова.*)
	resetAlarms: BOOL;		(*Сброс аварий насоса.*)
	delayRepeatedStartTime: WORD;		(*Количество секунд на задержку повторного пуска насоса.
Защита от частых включений. Если ничего не подключено = 300сек.*)
	alarmPump1input: BOOL;		(*Вход от источника сигнала об аварии насоса 1.*)
	alarmPump2input: BOOL;		(*Вход от источника сигнала об аварии насоса 2.*)
	driveAlarm: BOOL;		(*Сигнал авария от ЧРП.*)
END_VAR
VAR_OUTPUT
	regimePump1Main: BOOL;		(*Текущий режим - насос 1 = главный.*)
	regimePump2Main: BOOL;		(*Текущий режим - насос 2 = главный.*)
	regimeByCounter: BOOL;		(*Текущий режим - по количеству включений.*)
	regimeByWorkTime: BOOL;		(*Текущий режим - по наработке.*)
	counterPump1: DWORD;		(*Количество включений насоса 1.*)
	counterPump2: DWORD;		(*Количество включений насоса 2.*)
	daysPump1: WORD;		(*Количество отработанных дней насоса 1.*)
	hoursPump1: WORD;		(*Количество отработанных часов насоса 1.*)
	minutesPump1: WORD;		(*Количество отработанных минут насоса 1.*)
	secondsPump1: WORD;		(*Количество отработанных секунд насоса 1.*)
	daysPump2: WORD;		(*Количество отработанных дней насоса 2.*)
	hoursPump2: WORD;		(*Количество отработанных часов насоса 2.*)
	minutesPump2: WORD;		(*Количество отработанных минут насоса 2.*)
	secondsPump2: WORD;		(*Количество отработанных секунд насоса 2.*)
	drivePower: BOOL;		(*Сигнал на включение контактора частотного преобразователя.*)
	pump1ON: BOOL;		(*Сигнал на включение контактора насоса 1.*)
	pump2ON: BOOL;		(*Сигнал на включение контактора насоса 2.*)
	startDrive: BOOL;		(*Сигнал на запуск в частотный преобразователь.*)
	nextStartP1timer: WORD;		(*Обратный отсчет до возможности повторного пуска насоса 1.*)
	nextStartP2timer: WORD;		(*Обратный отсчет до возможности повторного пуска насоса 2.*)
	alarmPump1output: BOOL;		(*Сигнал авария насоса 1.
Триггерится, нужен сброс.*)
	alarmPump2output: BOOL;		(*Сигнал авария насоса 2.
Триггерится, нужен сброс.*)
END_VAR
VAR

	RichTwoPumpManager: RichTwoPumpManager;		(*Блок управления двумя насосами.*)
	TwoPumpOneDriveModule: TwoPumpOneDriveModule;		(*Модуль управления контакторами двух насосов и питания одного частотного преобразователя.*)
END_VAR
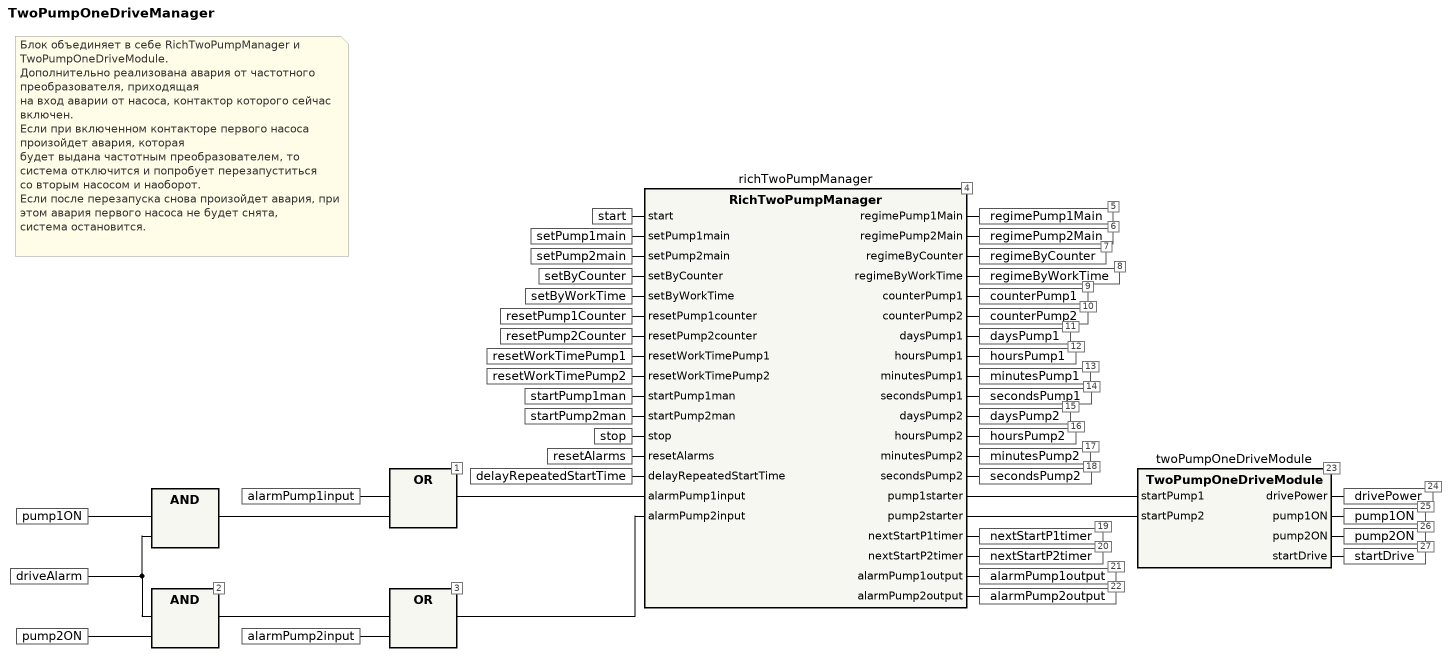
_CFC_ (* Continuous Function Chart, elements in execution order *)
(* Блок объединяет в себе RichTwoPumpManager и TwoPumpOneDriveModule. / Дополнительно реализована авария от частотного преобразователя, приходящая / на вход аварии от насоса, контактор которого сейчас включен. / Если при включенном контакторе первого насоса произойдет авария, которая / будет выдана частотным преобразователем, то система отключится и попробует перезапуститься / со вторым насосом и наоборот. / Если после перезапуска снова произойдет авария, при этом авария первого насоса не будет снята, / система остановится. *)
#0 AND(pump1ON, driveAlarm)
#1 OR(alarmPump1input, #0)
#2 AND(driveAlarm, pump2ON)
#3 OR(#2, alarmPump2input)
#4 richTwoPumpManager:RichTwoPumpManager(start: start, setPump1main: setPump1main, setPump2main: setPump2main, setByCounter: setByCounter, setByWorkTime: setByWorkTime, resetPump1counter: resetPump1Counter, resetPump2counter: resetPump2Counter, resetWorkTimePump1: resetWorkTimePump1, resetWorkTimePump2: resetWorkTimePump2, startPump1man: startPump1man, startPump2man: startPump2man, stop: stop, resetAlarms: resetAlarms, delayRepeatedStartTime: delayRepeatedStartTime, alarmPump1input: #1, alarmPump2input: #3)
#5 regimePump1Main <= #4.regimePump1Main
#6 regimePump2Main <= #4.regimePump2Main
#7 regimeByCounter <= #4.regimeByCounter
#8 regimeByWorkTime <= #4.regimeByWorkTime
#9 counterPump1 <= #4.counterPump1
#10 counterPump2 <= #4.counterPump2
#11 daysPump1 <= #4.daysPump1
#12 hoursPump1 <= #4.hoursPump1
#13 minutesPump1 <= #4.minutesPump1
#14 secondsPump1 <= #4.secondsPump1
#15 daysPump2 <= #4.daysPump2
#16 hoursPump2 <= #4.hoursPump2
#17 minutesPump2 <= #4.minutesPump2
#18 secondsPump2 <= #4.secondsPump2
#19 nextStartP1timer <= #4.nextStartP1timer
#20 nextStartP2timer <= #4.nextStartP2timer
#21 alarmPump1output <= #4.alarmPump1output
#22 alarmPump2output <= #4.alarmPump2output
#23 twoPumpOneDriveModule:TwoPumpOneDriveModule(startPump1: #4.pump1starter, startPump2: #4.pump2starter)
#24 drivePower <= #23.drivePower
#25 pump1ON <= #23.pump1ON
#26 pump2ON <= #23.pump2ON
#27 startDrive <= #23.startDrive
_END_CFC_
(* the same logic as Structured Text *)
(* Блок объединяет в себе RichTwoPumpManager и TwoPumpOneDriveModule. / Дополнительно реализована авария от частотного преобразователя, приходящая / на вход аварии от насоса, контактор которого сейчас включен. / Если при включенном контакторе первого насоса произойдет авария, которая / будет выдана частотным преобразователем, то система отключится и попробует перезапуститься / со вторым насосом и наоборот. / Если после перезапуска снова произойдет авария, при этом авария первого насоса не будет снята, / система остановится. *)
richTwoPumpManager(start := start, setPump1main := setPump1main, setPump2main := setPump2main, setByCounter := setByCounter, setByWorkTime := setByWorkTime, resetPump1counter := resetPump1Counter, resetPump2counter := resetPump2Counter, resetWorkTimePump1 := resetWorkTimePump1, resetWorkTimePump2 := resetWorkTimePump2, startPump1man := startPump1man, startPump2man := startPump2man, stop := stop, resetAlarms := resetAlarms, delayRepeatedStartTime := delayRepeatedStartTime, alarmPump1input := alarmPump1input OR (pump1ON AND driveAlarm), alarmPump2input := (driveAlarm AND pump2ON) OR alarmPump2input);
regimePump1Main := richTwoPumpManager.regimePump1Main;
regimePump2Main := richTwoPumpManager.regimePump2Main;
regimeByCounter := richTwoPumpManager.regimeByCounter;
regimeByWorkTime := richTwoPumpManager.regimeByWorkTime;
counterPump1 := richTwoPumpManager.counterPump1;
counterPump2 := richTwoPumpManager.counterPump2;
daysPump1 := richTwoPumpManager.daysPump1;
hoursPump1 := richTwoPumpManager.hoursPump1;
minutesPump1 := richTwoPumpManager.minutesPump1;
secondsPump1 := richTwoPumpManager.secondsPump1;
daysPump2 := richTwoPumpManager.daysPump2;
hoursPump2 := richTwoPumpManager.hoursPump2;
minutesPump2 := richTwoPumpManager.minutesPump2;
secondsPump2 := richTwoPumpManager.secondsPump2;
nextStartP1timer := richTwoPumpManager.nextStartP1timer;
nextStartP2timer := richTwoPumpManager.nextStartP2timer;
alarmPump1output := richTwoPumpManager.alarmPump1output;
alarmPump2output := richTwoPumpManager.alarmPump2output;
twoPumpOneDriveModule(startPump1 := richTwoPumpManager.pump1starter, startPump2 := richTwoPumpManager.pump2starter);
drivePower := twoPumpOneDriveModule.drivePower;
pump1ON := twoPumpOneDriveModule.pump1ON;
pump2ON := twoPumpOneDriveModule.pump2ON;
startDrive := twoPumpOneDriveModule.startDrive;
END_FUNCTION_BLOCK

(* POU TwoPumpOneDriveModule, CFC *)
FUNCTION_BLOCK TwoPumpOneDriveModule
VAR_INPUT
	startPump1: BOOL;		(*Входящий сигнал на запуск первого насоса.*)
	startPump2: BOOL;		(*Входящий сигнал на запуск второго насоса.*)
END_VAR
VAR_OUTPUT
	drivePower: BOOL;		(*Выход управления контактором питания ЧРП.*)
	pump1ON: BOOL;		(*Выход управления контактором питания насоса 1.*)
	pump2ON: BOOL;		(*Выход управления контактором питания насоса 2.*)
	startDrive: BOOL;		(*Сигнал пуск в ЧРП.*)
END_VAR
VAR
	pump1Off: BOOL;		(*Сигнал на отключение контактора насоса 1.*)
	pump2Off: BOOL;		(*Сигнал на отключение контактора насоса 2.*)
	startP1trig: R_TRIG;		(*Триггер переднего фронта сигнала на запуск насоса 1.*)
	startP2trig: R_TRIG;		(*Триггер переднего фронта сигнала на запуск насоса 2.*)
	ifP1on: IfBOOL;		(*Блок отправляет сигнал на запуск насоса 1 по одной
			из двух веток в зависимости от состояния ключа.*)
	ifP2on: IfBOOL;		(*Блок отправляет сигнал на запуск насоса 2 по одной
			из двух веток в зависимости от состояния ключа.*)
	startDriveDelay: TON;		(*Блок задержки подачи сигнала на включение ЧРП.*)
	stopDriveTrig: F_TRIG;		(*Триггер спада сигнала на включение насоса 1 или 2 для
			снятия сигнала пуск в ЧРП.*)
	p1ONdelay: TON;		(*Задержка на включение контактора насоса 1.*)
	p2ONdelay: TON;		(*Задержка на включение контактора насоса 2.*)
	startDriveTrig: RS;		(*RS триггер сигнала пуск в ЧРП.*)
	p1powerTrig: RS;		(*RS триггер включения контактора насоса 1.*)
	p2powerTrig: RS;		(*RS триггер включения контактора насоса 2.*)
	offP1delayTrig: RS;		(*RS триггер сигнала на отключение контактора насоса 1.*)
	offP2delayTrig: RS;		(*RS триггер сигнала на отключение контактора насоса 2.*)
	offPowerDelay: TOF;		(*Блок управления временем выключения контактора питания ЧРП.*)
	offP2delay: TON;		(*Задержка выключения контактора насоса 1.*)
	offP1delay: TON;		(*Задержка выключения контактора насоса 2.*)
	fastStart: BOOL;		(*Быстрый сигнал на пуск в ЧРП, если не надо переключать
			контакторы.*)
END_VAR
VAR (* helpers for the ST form of the networks *)
	_t160 : BOOL;
END_VAR
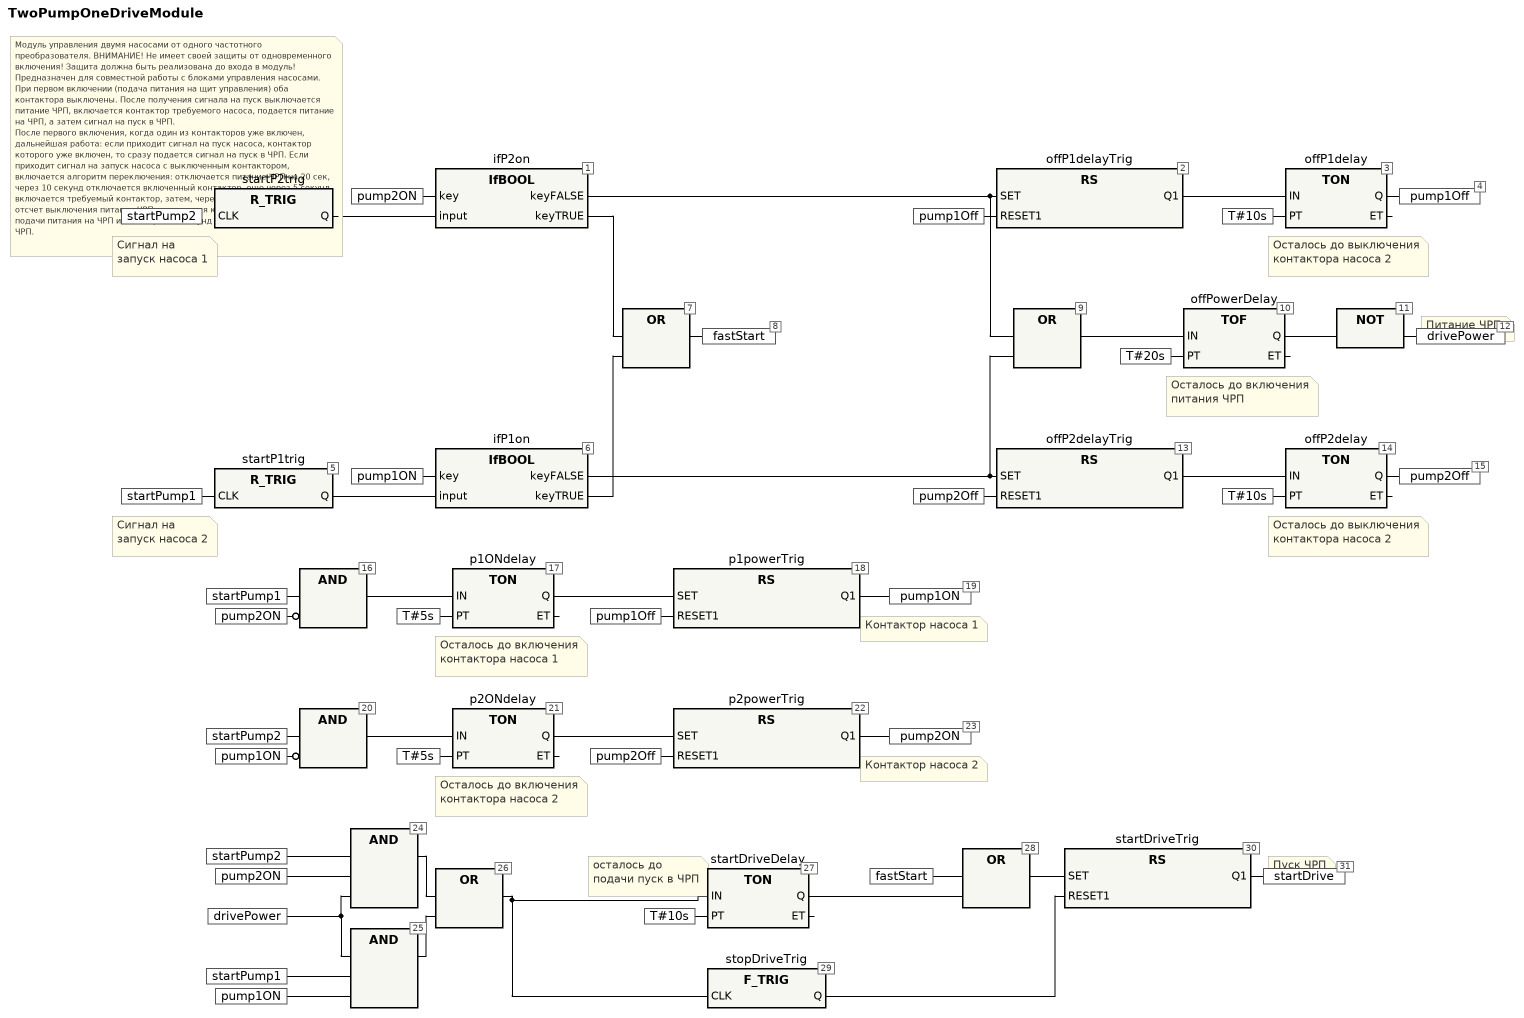
_CFC_ (* Continuous Function Chart, elements in execution order *)
(* Модуль управления двумя насосами от одного частотного преобразователя. ВНИМАНИЕ! Не имеет своей защиты от одновременного включения! Защита должна быть реализована до входа в модуль! Предназначен для совместной работы с блоками управления насосами. / При первом включении (подача питания на щит управления) оба контактора выключены. После получения сигнала на пуск выключается питание ЧРП, включается контактор требуемого насоса, подается питание на ЧРП, а затем сигнал на пуск в ЧРП. / После первого включения, когда один из контакторов уже включен, дальнейшая работа: если приходит сигнал на пуск насоса, контактор которого уже включен, то сразу подается сигнал на пуск в ЧРП. Если приходит сигнал на запуск насоса с выключенным контактором, / включается алгоритм переключения: отключается питание ЧРП на 20 сек, через 10 секунд отключается включенный контактор, еще через 5 секунд включается требуемый контактор, затем, через 5 секунд, заканчивается отсчет выключения питания ЧРП, включается контактор / подачи питания на ЧРП и еще через 10 секунд подается питание на пуск в ЧРП. *)
(* Сигнал на / запуск насоса 2 *)
(* Сигнал на / запуск насоса 1 *)
(* Контактор насоса 1 *)
(* Осталось до включения / контактора насоса 1 *)
(* Контактор насоса 2 *)
(* Осталось до выключения / контактора насоса 2 *)
(* Осталось до включения / питания ЧРП *)
(* Питание ЧРП. *)
(* Осталось до включения / контактора насоса 2 *)
(* Осталось до выключения / контактора насоса 2 *)
(* осталось до / подачи пуск в ЧРП *)
(* Пуск ЧРП *)
#0 startP2trig:R_TRIG(CLK: startPump2)
#1 ifP2on:IfBOOL(key: pump2ON, input: #0.Q)
#2 offP1delayTrig:RS(SET: #1.keyFALSE, RESET1: pump1Off)
#3 offP1delay:TON(IN: #2.Q1, PT: T#10s)
#4 pump1Off <= #3.Q
#5 startP1trig:R_TRIG(CLK: startPump1)
#6 ifP1on:IfBOOL(key: pump1ON, input: #5.Q)
#7 OR(#1.keyTRUE, #6.keyTRUE)
#8 fastStart <= #7
#9 OR(#1.keyFALSE, #6.keyFALSE)
#10 offPowerDelay:TOF(IN: #9, PT: T#20s)
#11 NOT(#10.Q)
#12 drivePower <= #11
#13 offP2delayTrig:RS(SET: #6.keyFALSE, RESET1: pump2Off)
#14 offP2delay:TON(IN: #13.Q1, PT: T#10s)
#15 pump2Off <= #14.Q
#16 AND(startPump1, NOT pump2ON)
#17 p1ONdelay:TON(IN: #16, PT: T#5s)
#18 p1powerTrig:RS(SET: #17.Q, RESET1: pump1Off)
#19 pump1ON <= #18.Q1
#20 AND(startPump2, NOT pump1ON)
#21 p2ONdelay:TON(IN: #20, PT: T#5s)
#22 p2powerTrig:RS(SET: #21.Q, RESET1: pump2Off)
#23 pump2ON <= #22.Q1
#24 AND(startPump2, pump2ON, drivePower)
#25 AND(drivePower, startPump1, pump1ON)
#26 OR(#24, #25)
#27 startDriveDelay:TON(IN: #26, PT: T#10s)
#28 OR(fastStart, #27.Q)
#29 stopDriveTrig:F_TRIG(CLK: #26)
#30 startDriveTrig:RS(SET: #28, RESET1: #29.Q)
#31 startDrive <= #30.Q1
_END_CFC_
(* the same logic as Structured Text *)
(* Модуль управления двумя насосами от одного частотного преобразователя. ВНИМАНИЕ! Не имеет своей защиты от одновременного включения! Защита должна быть реализована до входа в модуль! Предназначен для совместной работы с блоками управления насосами. / При первом включении (подача питания на щит управления) оба контактора выключены. После получения сигнала на пуск выключается питание ЧРП, включается контактор требуемого насоса, подается питание на ЧРП, а затем сигнал на пуск в ЧРП. / После первого включения, когда один из контакторов уже включен, дальнейшая работа: если приходит сигнал на пуск насоса, контактор которого уже включен, то сразу подается сигнал на пуск в ЧРП. Если приходит сигнал на запуск насоса с выключенным контактором, / включается алгоритм переключения: отключается питание ЧРП на 20 сек, через 10 секунд отключается включенный контактор, еще через 5 секунд включается требуемый контактор, затем, через 5 секунд, заканчивается отсчет выключения питания ЧРП, включается контактор / подачи питания на ЧРП и еще через 10 секунд подается питание на пуск в ЧРП. *)
(* Сигнал на / запуск насоса 2 *)
(* Сигнал на / запуск насоса 1 *)
(* Контактор насоса 1 *)
(* Осталось до включения / контактора насоса 1 *)
(* Контактор насоса 2 *)
(* Осталось до выключения / контактора насоса 2 *)
(* Осталось до включения / питания ЧРП *)
(* Питание ЧРП. *)
(* Осталось до включения / контактора насоса 2 *)
(* Осталось до выключения / контактора насоса 2 *)
(* осталось до / подачи пуск в ЧРП *)
(* Пуск ЧРП *)
startP2trig(CLK := startPump2);
ifP2on(key := pump2ON, input := startP2trig.Q);
offP1delayTrig(SET := ifP2on.keyFALSE, RESET1 := pump1Off);
offP1delay(IN := offP1delayTrig.Q1, PT := T#10s);
pump1Off := offP1delay.Q;
startP1trig(CLK := startPump1);
ifP1on(key := pump1ON, input := startP1trig.Q);
fastStart := ifP2on.keyTRUE OR ifP1on.keyTRUE;
offPowerDelay(IN := ifP2on.keyFALSE OR ifP1on.keyFALSE, PT := T#20s);
drivePower := NOT offPowerDelay.Q;
offP2delayTrig(SET := ifP1on.keyFALSE, RESET1 := pump2Off);
offP2delay(IN := offP2delayTrig.Q1, PT := T#10s);
pump2Off := offP2delay.Q;
p1ONdelay(IN := startPump1 AND NOT pump2ON, PT := T#5s);
p1powerTrig(SET := p1ONdelay.Q, RESET1 := pump1Off);
pump1ON := p1powerTrig.Q1;
p2ONdelay(IN := startPump2 AND NOT pump1ON, PT := T#5s);
p2powerTrig(SET := p2ONdelay.Q, RESET1 := pump2Off);
pump2ON := p2powerTrig.Q1;
_t160 := (startPump2 AND pump2ON AND drivePower) OR (drivePower AND startPump1 AND pump1ON);
startDriveDelay(IN := _t160, PT := T#10s);
stopDriveTrig(CLK := _t160);
startDriveTrig(SET := fastStart OR startDriveDelay.Q, RESET1 := stopDriveTrig.Q);
startDrive := startDriveTrig.Q1;
END_FUNCTION_BLOCK
